INTERFACE ITFMotor

METHOD Aan
VAR_INPUT
END_VAR
END_METHOD

PROPERTY MotorStatus : EMotorStatus
GET
END_GET
SET
END_SET
END_PROPERTY

METHOD Uit
VAR_INPUT
END_VAR
END_METHOD

END_INTERFACE

(* stored: Version 1.1.0.1
   Itf ITFMotor: Id {d3f47777-bd5b-48b1-bdcb-ea49bd88495e}
   Method Aan: Id {060d63f9-787c-496d-9022-28764b8b1e72}
   Property MotorStatus: Id {74bf9a58-abad-4fd1-b45d-2376d0b9f086}
   Get Get: Id {cbbdf476-21d7-4c49-b33e-149823c47cf1}
   Set Set: Id {d4e3075b-24cb-4947-8d59-d54dd0417254}
   Method Uit: Id {123d9254-67f0-4f43-bd52-c35d6297472c} *)
